// TIA Portal project "vize" (V15.1)

(* hardware
DEVICE "S7-1200 station_1"  S7-1200 Station
   slot 0: "Rack_0"  S7-1200 Rack  Rack  V1.0
   slot 1: "PLC_1"  CPU 1214C DC/DC/DC  6ES7 214-1AG40-0XB0  V4.2
*)

// ===== PLC "PLC_1"  CPU 1214C DC/DC/DC =====

VAR_GLOBAL   // PLC tag table "Default tag table"
   "General_Start" AT %M0.0 : Bool;
   "Reset_and_Start" AT %Q0.0 : Bool;
   "Start_Control_Loop" AT %Q0.1 : Bool;
   "Time_End" AT %M0.1 : Bool;
END_VAR

DATA_BLOCK "general_memory"   // DB1
{ S7_Optimized_Access := 'TRUE' }
VERSION : 0.1
   VAR RETAIN
      x1_data : Array[0..200] of Real;
      x2_data : Array[0..200] of Real;
      u_data : Array[0..200] of Real;
   END_VAR
BEGIN
END_DATA_BLOCK

DATA_BLOCK "Initial_values_DB"   // DB2
{ S7_Optimized_Access := 'TRUE' }
VERSION : 0.1
// stored: InstanceOfName Initial_values
"Initial_values"
BEGIN
END_DATA_BLOCK

DATA_BLOCK "System_Integration_DB"   // DB4
{ S7_Optimized_Access := 'TRUE' }
VERSION : 0.1
// stored: InstanceOfName System_Integration
"System_Integration"
BEGIN
END_DATA_BLOCK

// folder: System blocks/Program resources

DATA_BLOCK "General_Timer"   // DB3
{ S7_Optimized_Access := 'TRUE' }
AUTHOR : Simatic
FAMILY : IEC
NAME : IEC_TMR
VERSION : 1.0
// stored: InstanceOfName IEC_TIMER
"IEC_TIMER"
BEGIN
END_DATA_BLOCK

// folder: (top level)

FUNCTION_BLOCK "Initial_values"   // FB1, LAD
{ S7_Optimized_Access := 'TRUE' }
VERSION : 0.1
   VAR_INPUT
      start : Bool;
   END_VAR
BEGIN

REGION Network 1
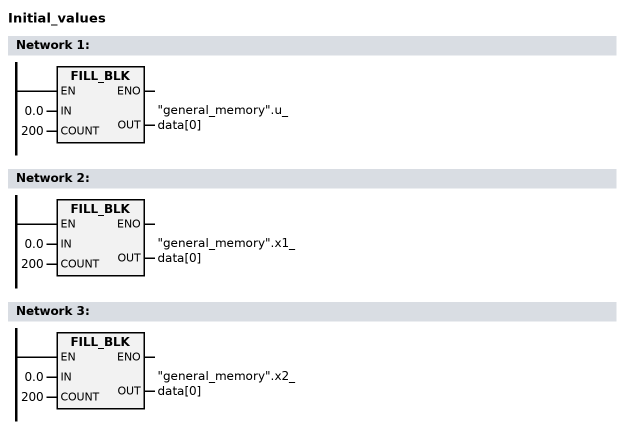
   RUNG wire#powerrail
      FillBlockI(in := 0.0, count := 200, out => "general_memory".u_data[0])
   END_RUNG
   // the same network as SCL:
   FILL_BLK(IN := 0.0, COUNT := 200, OUT => "general_memory".u_data[0]);
END_REGION

REGION Network 2
   RUNG wire#powerrail
      FillBlockI(in := 0.0, count := 200, out => "general_memory".x1_data[0])
   END_RUNG
   // the same network as SCL:
   FILL_BLK(IN := 0.0, COUNT := 200, OUT => "general_memory".x1_data[0]);
END_REGION

REGION Network 3
   RUNG wire#powerrail
      FillBlockI(in := 0.0, count := 200, out => "general_memory".x2_data[0])
   END_RUNG
   // the same network as SCL:
   FILL_BLK(IN := 0.0, COUNT := 200, OUT => "general_memory".x2_data[0]);
END_REGION
END_FUNCTION_BLOCK

FUNCTION_BLOCK "System_Integration"   // FB2, LAD
{ S7_Optimized_Access := 'TRUE' }
VERSION : 0.1
   VAR_INPUT
      Start_Control_Loop : Bool;
   END_VAR
   VAR
      pozitif_kenar : Bool;
      k : Int;
      x1temp : Real;
      x2temp : Real;
      xref1 : Real;
      xref2 : Real;
      xref1new : Real;
      xref2new : Real;
      ww_cos : Real;
      error1 : Real;
      error2 : Real;
      surface : Real;
      "abs(surface)" : Real;
      sat : Real;
      tan_op : Real;
      fhat : Real;
      dot_deriv : Real;
      uk : Real;
      minus_fhat : Real;
      x1_new : Real;
      x2_new : Real;
   END_VAR
   VAR_TEMP   // added for the SCL form of the ladder/FBD networks
      _w1 : Bool;
   END_VAR
BEGIN

REGION Network 1
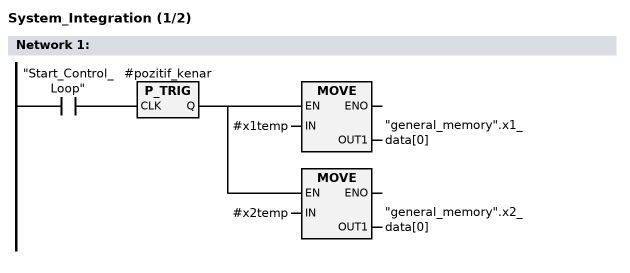
   RUNG wire#powerrail
      Contact( "Start_Control_Loop" )
      P_Trig( #pozitif_kenar )
      wire#w1
      Move(in := #x1temp, out1 => "general_memory".x1_data[0])
   END_RUNG
   RUNG wire#w1
      Move(in := #x2temp, out1 => "general_memory".x2_data[0])
   END_RUNG
   // the same network as SCL:
   #_w1 := "Start_Control_Loop" AND NOT #pozitif_kenar;   // rising edge
   #pozitif_kenar := "Start_Control_Loop";
   IF #_w1 THEN
       "general_memory".x1_data[0] := #x1temp;
       "general_memory".x2_data[0] := #x2temp;
   END_IF;
END_REGION

REGION Network 2
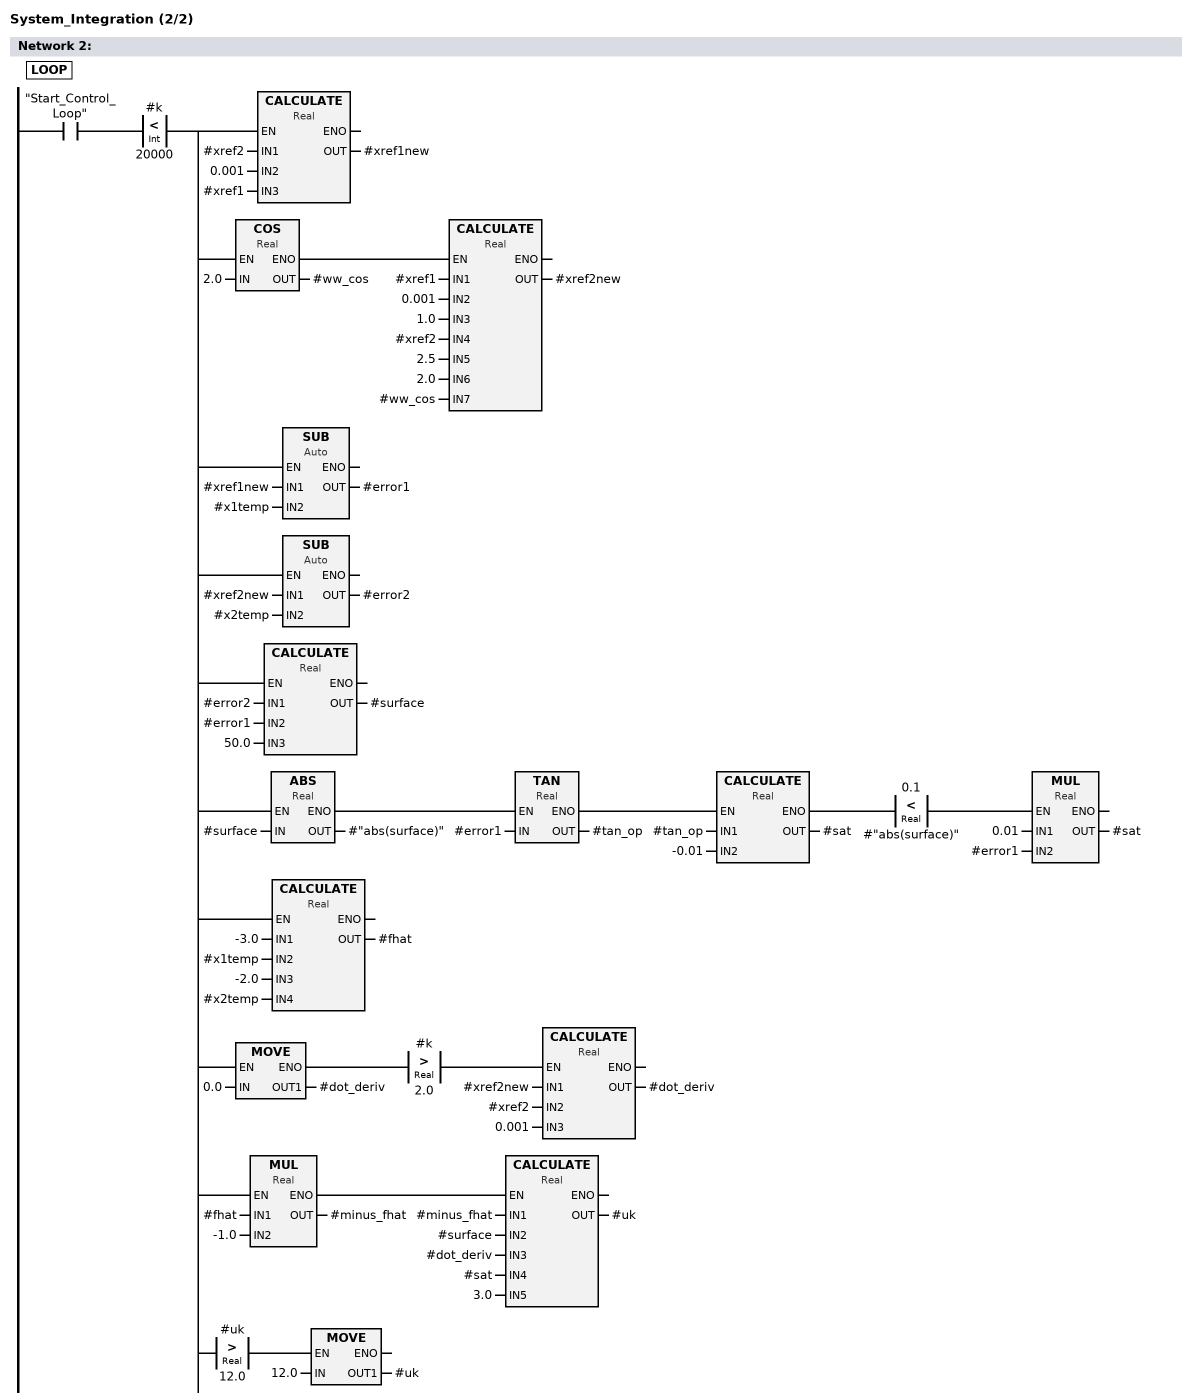
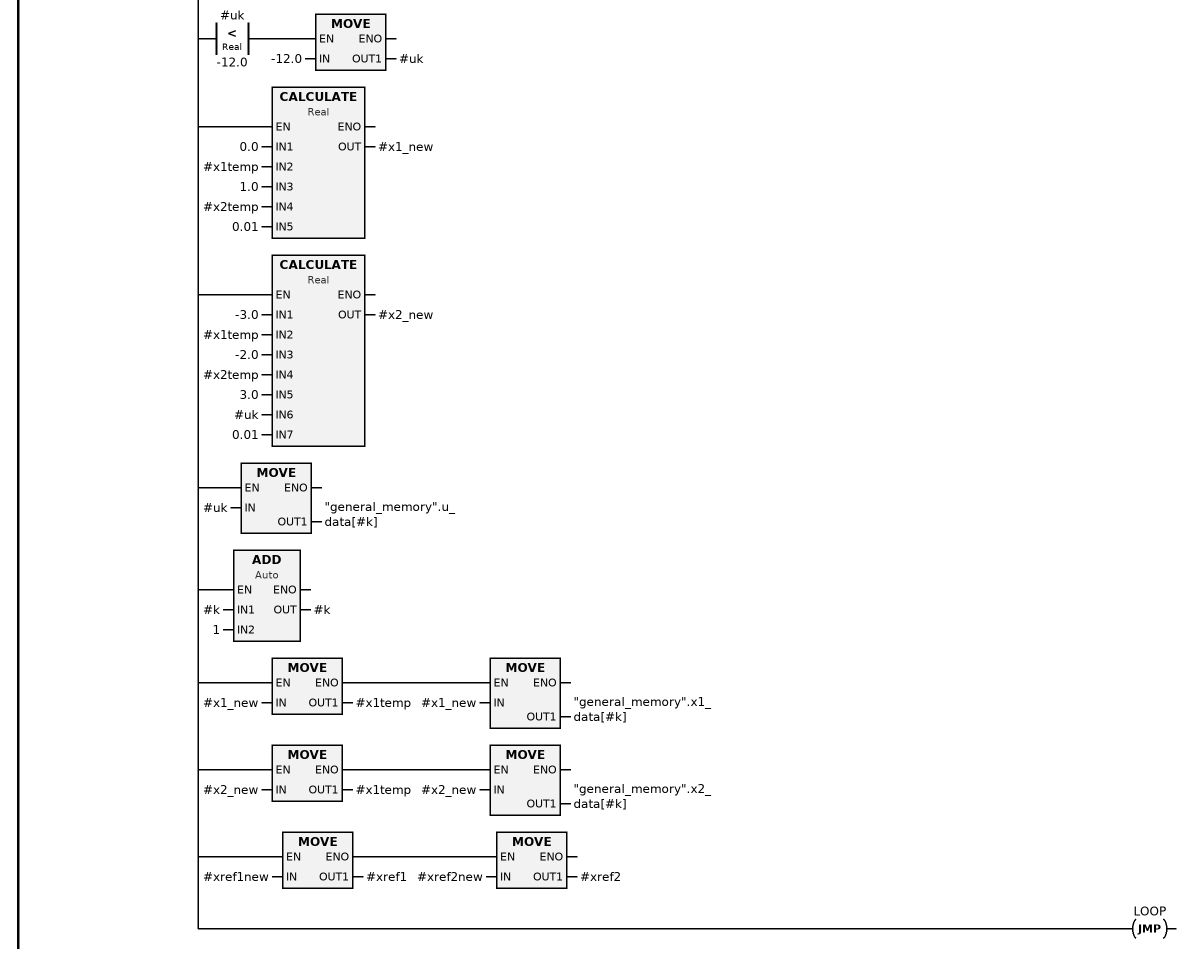
   LOOP:
   #_w1 := "Start_Control_Loop" AND (#k < 20000);
   IF #_w1 THEN
       #xref1new := #xref2*0.001+#xref1;
       #ww_cos := COS(2.0);
       #xref2new := #xref1+0.001*(1.0*(1.0-#xref1**2.0)*#xref2-#xref1+2.5*#ww_cos);
       #error1 := #xref1new - #x1temp;
       #error2 := #xref2new - #x2temp;
       #surface := #error2+#error1*50.0;
       #"abs(surface)" := ABS(#surface);
       #tan_op := TAN(#error1);
       #sat := #tan_op*(-0.01);
   END_IF;
   IF #_w1 AND (0.1 < #"abs(surface)") THEN #sat := 0.01 * #error1; END_IF;
   IF #_w1 THEN
       #fhat := (-3.0)*#x1temp+(-2.0)*#x2temp;
       #dot_deriv := 0.0;
   END_IF;
   IF #_w1 AND (#k > 2.0) THEN #dot_deriv := (#xref2new-#xref2)/0.001; END_IF;
   IF #_w1 THEN
       #minus_fhat := #fhat * (-1.0);
       #uk := (#minus_fhat+#surface+#dot_deriv+#sat)/3.0;
   END_IF;
   IF #_w1 AND (#uk > 12.0) THEN #uk := 12.0; END_IF;
   IF #_w1 AND (#uk < (-12.0)) THEN #uk := -12.0; END_IF;
   IF #_w1 THEN
       #x1_new := #x1temp+0.01*(0.0*#x1temp+1.0*#x2temp);
       #x2_new := #x2temp+0.01*((-3.0)*#x1temp+(-2.0)*#x2temp+3.0*#uk);
       "general_memory".u_data[#k] := #uk;
       #k := #k + 1;
       #x1temp := #x1_new;
       "general_memory".x1_data[#k] := #x1_new;
       #x1temp := #x2_new;
       "general_memory".x2_data[#k] := #x2_new;
       #xref1 := #xref1new;
       #xref2 := #xref2new;
       GOTO LOOP;
   END_IF;
END_REGION
END_FUNCTION_BLOCK

ORGANIZATION_BLOCK "Main"   // OB1, LAD, ProgramCycle
TITLE = "Main Program Sweep (Cycle)"
{ S7_Optimized_Access := 'TRUE' }
VERSION : 0.1
   VAR_INPUT
      Initial_Call : Bool;   // Initial call of this OB
      Remanence : Bool;   // =True, if remanent data are available
   END_VAR
   VAR_TEMP   // added for the SCL form of the ladder/FBD networks
      _w1 : Bool;
   END_VAR
BEGIN

REGION Network 1
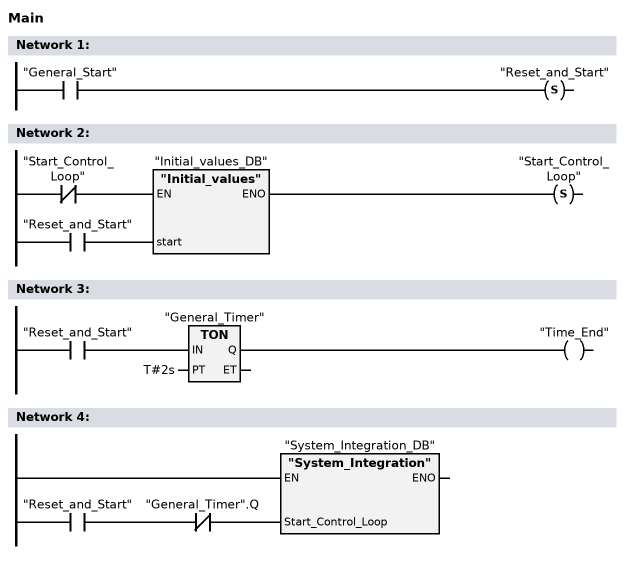
   RUNG wire#powerrail
      Contact( "General_Start" )
      S_Coil( "Reset_and_Start" )
   END_RUNG
   // the same network as SCL:
   IF "General_Start" THEN "Reset_and_Start" := TRUE; END_IF;
END_REGION

REGION Network 2
   RUNG wire#powerrail
      I_Contact( "Start_Control_Loop" )
      "Initial_values_DB"(start := wire#w1)
      S_Coil( "Start_Control_Loop" )
   END_RUNG
   RUNG wire#powerrail
      Contact( "Reset_and_Start" )
   END_RUNG wire#w1
   // the same network as SCL:
   "Initial_values_DB"(EN := NOT "Start_Control_Loop", start := "Reset_and_Start", ENO => #_w1);   // "Initial_values"
   IF #_w1 THEN "Start_Control_Loop" := TRUE; END_IF;
END_REGION

REGION Network 3
   "General_Timer".TON(IN := "Reset_and_Start", PT := T#2s);
   "Time_End" := "General_Timer".Q;
END_REGION

REGION Network 4
   RUNG wire#powerrail
      "System_Integration_DB"(Start_Control_Loop := wire#w1)
   END_RUNG
   RUNG wire#powerrail
      Contact( "Reset_and_Start" )
      I_Contact( "General_Timer".Q )
   END_RUNG wire#w1
   // the same network as SCL:
   "System_Integration_DB"(Start_Control_Loop := "Reset_and_Start" AND NOT "General_Timer".Q);   // "System_Integration"
END_REGION
END_ORGANIZATION_BLOCK